{attribute 'GeneratedUsingTerminal: IODEVICETYPE_ETHERCATPROT'}
{attribute addProperty BoxType "IODEVICETYPE_ETHERCATPROT"}
{attribute addProperty Id "WcStateAT %I*WcState_0B2B16F91InfoDataAT %I*InfoData_8649EEEB8"}
{attribute addProperty CRC "2872004729"}
{attribute addProperty Size "9"}
TYPE SyncUnitTask_AB2F5079 EXTENDS SyncUnitTaskBase_FCD3CBF3 :
STRUCT
	{attribute addProperty Name "WcState"}
	WcState : WcState_0B2B16F9;
	{attribute addProperty Name "InfoData"}
	InfoData : InfoData_8649EEEB;
END_STRUCT
END_TYPE

(* stored: Version 1.1.0.1, ProductVersion 3.1.4024.12
   DUT SyncUnitTask_AB2F5079: Id {b2b590df-e754-0551-0b33-f0a985b90142} *)
